// TIA Portal V21 export
// export: Created 2026-09-06T16:30:00Z, ExportSetting WithDefaults
FUNCTION "FC_LAD_Test" : Void   // FC20, LAD
{ S7_Optimized_Access := 'TRUE' }
VERSION : 0.1
// stored: AutoNumber true, SetENOAutomatically false
BEGIN

REGION Network 1: Teste LAD START para H2
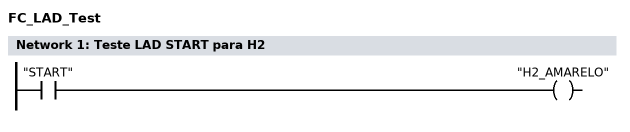
   RUNG wire#powerrail
      Contact( "START" )
      Coil( "H2_AMARELO" )
   END_RUNG
   // the same network as SCL:
   "H2_AMARELO" := "START";
END_REGION
END_FUNCTION
